// TIA Portal V18 export
FUNCTION "CheckData" : Void   // FC4023, SCL
{ S7_Optimized_Access := 'FALSE' }
// stored: AutoNumber false, SetENOAutomatically false
   VAR_INPUT
      DBNo : Int;
      DBBNO : Int;
      ByteLenth : Int;
   END_VAR
   VAR_OUTPUT
      AlarmON : Bool;
   END_VAR
   VAR_TEMP
      AlarmByte : Int;
      tByte : Int;
   END_VAR
BEGIN
   #AlarmON := 0;
   #AlarmByte := 0;
   IF #ByteLenth>0 THEN
       FOR #tByte:=0 TO #ByteLenth-1 DO
           IF PEEK_BYTE(area:=16#84,dbNumber:=#DBNo,byteOffset:=#DBBNO+#tByte)<>0 THEN
               #AlarmON := TRUE;
               #AlarmByte := #DBBNO + #tByte;
               EXIT;
           ELSE
               #AlarmON := false;
               #AlarmByte := 0;
           END_IF;
       END_FOR;
   END_IF;
END_FUNCTION
